RoboDK station: Pickup Piece, Stitch Piece & Go Home.rdk

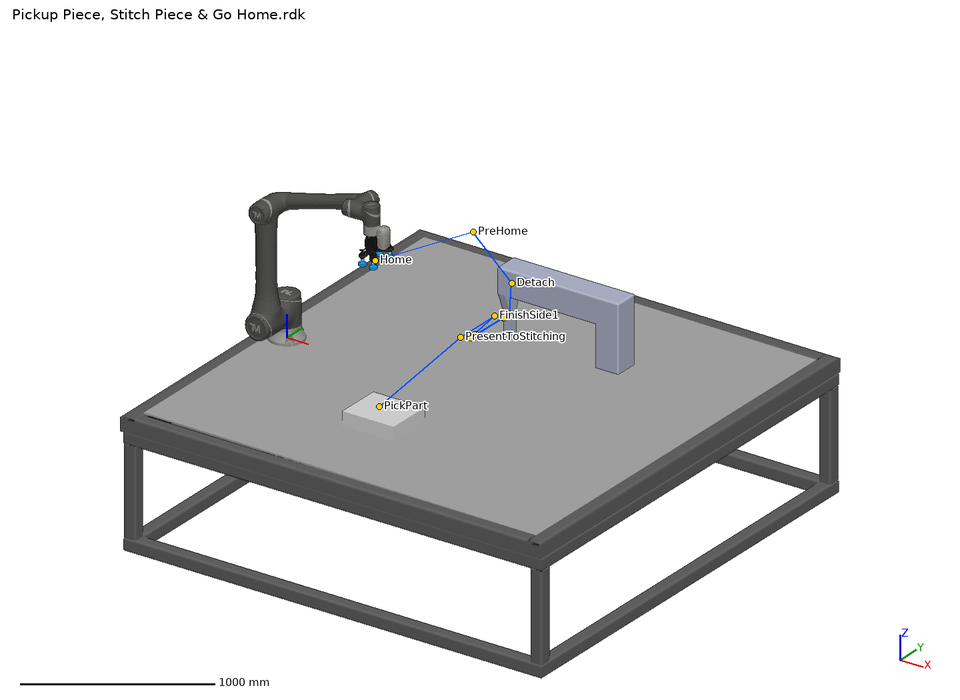
[picture v0: the station drawn from its stored meshes, robots at their saved joint values, targets as dots, program paths as lines]
Station STAR2 (saved by RoboDK 5.1.1). Poses are relative to the parent item; angles as X-Y-Z fixed-axis rotations.
  - frame Omron TM12 Base at (190, -120, 780) mm
    - robot Omron TM12: 6 axes, payload 12 kg, reach 1300 mm, repeatability 0.1 mm, weight 33.3 kg
        modified DH rows (alpha deg, a mm, theta deg, d mm): 0, 0, 0, 165.2; 90, 0, 90, 0; 0, 636.1, 0, 0; 0, 557.9, -90, 156.3; -90, 0, 0, 106; 90, 0, 180, 113.15
        joint limits [-270, -180, -166, -180, -180, -270] to [270, 180, 166, 180, 180, 270]; home [0, 0, 90, 0, 90, 0]; saved at [0, -0.459, 75.498, 14.96, 90, 0]
      - tool RobotiQ EPick Four Vacuum Cup, TCP at (0, 24, 144) mm, size 191.2 x 117.6 x 147.9 mm
    - target Home (Cartesian target) at (663.9, -156.3, 688.15) mm, rotated rx 180 ry 0 rz 90 deg; joints [0, -0.459, 75.498, 14.96, 90, 0] of Omron TM12
    - target PickPart (Cartesian target) at (950, -530, 84) mm, rotated rx -180 ry 0 rz 90 deg; joints [-21.361, 46.118, 72.239, -28.357, 90, -21.361] of Omron TM12
    - target PresentToStitching (Cartesian target) at (825, 375, 84) mm, rotated rx -180 ry 0 rz 90 deg; joints [35.266, 32.291, 98.135, -40.426, 90, 35.266] of Omron TM12
    - target FinishSide1 (Cartesian target) at (825, 680, 84) mm, rotated rx -180 ry 0 rz 90 deg; joints [48.884, 44.769, 74.84, -29.609, 90, 48.884] of Omron TM12
    - target StartSide2 (Cartesian target) at (868.34, 400.98, 84) mm, rotated rx -180 ry 0 rz 178.75 deg; joints [32.989, 36.713, 90.058, -36.772, 90, -55.761] of Omron TM12
    - target FinishSide2 (Cartesian target) at (873.9, 685.92, 84) mm, rotated rx 180 ry 0 rz 178.75 deg; joints [45.358, 48.613, 67.39, -26.004, 90, -43.392] of Omron TM12
    - target StartSide3 (Cartesian target) at (873.9, 450, 84) mm, rotated rx -180 ry 0 rz -90 deg; joints [35.572, 41.082, 81.878, -32.959, 90, -144.428] of Omron TM12
    - target FinishSide3 (Cartesian target) at (873.9, 690, 84) mm, rotated rx -180 ry 0 rz -90 deg; joints [45.475, 51.979, 60.784, -22.762, 90, -134.525] of Omron TM12
    - target StartSide4 (Cartesian target) at (868.44, 440.06, 84) mm, rotated rx -180 ry 0 rz -1.25 deg; joints [37.233, 39.611, 84.653, -34.264, 90, -231.517] of Omron TM12
    - target FinishSide4 (Cartesian target) at (874.99, 739.99, 84) mm, rotated rx -180 ry 0 rz -1.25 deg; joints [48.839, 54.939, 54.913, -19.852, 90, -219.911] of Omron TM12
    - target Detach (Cartesian target) at (676.58, 1044.39, 84) mm, rotated rx -180 ry 0 rz -1.25 deg; joints [64.733, 68.972, 26.406, -5.379, 90, -204.017] of Omron TM12
    - target PreHome (Cartesian target) at (572.24, 846.62, 424) mm, rotated rx -180 ry 0 rz -1.25 deg; joints [64.743, 35.128, 70.287, -15.415, 90, 155.993] of Omron TM12
  - object Table 108x114x32 IN at (0, 0, 0) mm, size 2628.9 x 2679.7 x 778.4 mm, geometry from Table-108x114x32-IN.sld
    - object Ventac at (1140, -650, 1004) mm, size 322.4 x 278.6 x 84.2 mm, geometry from Untitled-6012cee7.stl
  - program PicknPlace (21 instructions, listed below)
  - object Sweing Machine at (1770, 520, 860) mm, size 760 x 150 x 400 mm, geometry from Sweing Machine.IGS
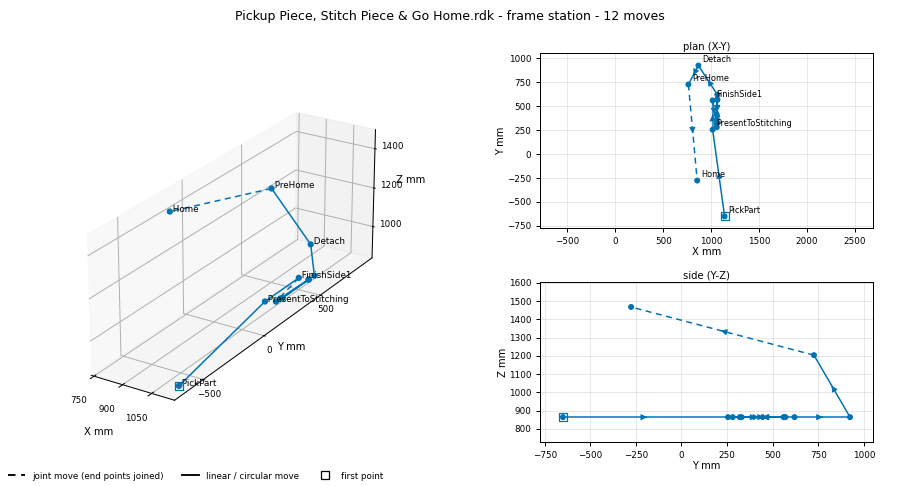
[picture p0: tool path of Pickup Piece, Stitch Piece & Go Home.rdk in frame station, 12 of 12 moves have a stored position in this frame; points joined in program order, loops and branches not executed]

--- program PicknPlace (robot Omron TM12) ---
  Set Ref.: Omron TM12 Base
  Accurate (rounding -1 mm)
  Set speed (150.0 mm/s)
  MoveJ (Target 1) -> target PickPart
  Attach to RobotiQ EPick Four Vacuum Cup
  MoveL (PresentToStitching)
  MoveL (FinishSide1)
  MoveJ (StartSide2)
  MoveL (FinishSide2)
  MoveJ (StartSide3)
  MoveL (FinishSide3)
  MoveJ (StartSide4)
  MoveL (FinishSide4)
  MoveL (Detach)
  Detach from RobotiQ EPick Four Vacuum Cup
  Smooth(3)
  MoveL (PreHome)
  MoveJ (Home)
  Replace Ventac
  Call Program1
  Not defined
